TYPE ST_ITC_ESR :
(**************************************************************************************
 * 	Application		:	BoxControl Framework
 *	Revision		:	$Revision: 404529 $
 *	Revision date	:	$Date: 2018-04-23 08:21:38 +0200 (Mo., 23 Apr 2018) $
 *	Last changed by	:	$Author: b7bolm $
 *	URL				:	$URL: http://almscdc.swisslog.com/repo/SWPD/Development/BoxControlFramework/20_Release/trunk/01_Software/BCF/BCF/JumpStart/20_Product/10_App/11_Com/10_Lib/10_Conv/11_ITC/01_DUTs/ST_ITC_ESR.TcDUT $
 *
 *	Purpose			:	ESR Structure
 *
 * ------------------------------------------------------------------------------------
 *	Copyright Swisslog [IP AG], Switzerland. All rights reserved.
 * 
 * ------------------------------------------------------------------------------------
 *	
 * 	Revision History: 
 *
 * 	VERSION			DATE			INITIALS			DESCRIPTION
 *	0.1				01.01.2001		swl					Example
 *
 **************************************************************************************)
STRUCT
	Position 			: STRING(Conveyor.POSITION_STRINGLENGTH); // 12 Digit SIS Location MM-GGG-EEEE-LLL 
	State				: E_PositionState; // 1 Digit State 
	Enabled				: BOOL; // 1 Digit State 
	ErrorState			: E_ErrorState; // 1 Digit Error State 
	ErrorCode			: E_ErrorConv; // 4 Digit Return Code 
	ErrorType			: E_ErrorType; // 1 Digit Error Type 
	ErrorInformation	: STRING(System.ERROR_PARAM_STRINGLENGTH); // 5 Chars Error Information 
	Variable			: DINT; // 4 Digit Variable 
	ReturnCode			: E_ErrorConv; // 4 Digit error code
END_STRUCT
END_TYPE

(* stored: Version 1.1.0.1, ProductVersion 3.1.4022.12
   DUT ST_ITC_ESR: Id {f5ecd9da-267b-4b7d-b5d7-8c2dc062fac2} *)
